(*
Casts I_Component as I_Receiver.
Returns:
- Ok - Success,
- Err.InvRef - Invalid reference,
- Err.Itf0 - Invalid interface,
- Err.NoMatch - Cast failed
*)
FUNCTION ICompToIRec : Result
VAR_INPUT
	iIn		: I_Component;
	iOut	: REFERENCE TO I_Receiver;
END_VAR

IF NOT __ISVALIDREF(iOut) THEN
	ICompToIRec := Err.InvRef;
	RETURN;
END_IF

IF iIn = 0 THEN
	ICompToIRec := Err.Itf0;
	RETURN;
END_IF

IF __QUERYINTERFACE(iIn, iOut) THEN
	ICompToIRec := Ok;
ELSE
	ICompToIRec := Err.NoMatch;
END_IF

END_FUNCTION

(* stored: Version 1.1.0.1
   POU ICompToIRec: Id {9a02776e-f8c4-45bc-8c18-325d7f2421cf}, SpecialFunc None *)
